(* IEC 61131-3 sources: C32_CAN/Source, 4 files *)

(* ---- ReadLocalODEntry.ST ---- *)
FUNCTION_BLOCK ReadLocalODEntry
VAR CONSTANT

    (* Definition of Data types *)
    SOO_DT_BYTE     : USINT := 1;
    SOO_DT_WORD     : USINT := 2;
    SOO_DT_DWORD    : USINT := 4;

    DEVICE          : USINT := 0;   (* Device 0: local device            *)

END_VAR

VAR_INPUT

    usiNetNumber_i  : USINT;        (* Netnumber: 0=CAN=, 1=CAN1         *)
    wIndex_i        : WORD;         (* Index to read                     *)
    bSubIndex_i     : BYTE;         (* SubIndex to read                  *)

END_VAR

VAR_OUTPUT

    dwData_o        : DWORD;        (* Data read from OD entry           *)
    usiDataType_o   : USINT;        (* DataType: 1=Byte, 2=Word, 4=Dword *)
    xSuccess_o      : BOOL;         (* TRUE if SDO was successful        *)
    wError_o        : WORD;
    dwErrorInfo_o   : DWORD;

END_VAR

VAR

    FB_CanSdoRead8  : CAN_SDO_READ8;

END_VAR

(*=========================================================================*)
(*      FUNCTIONBLOCK ReadLocalODEntry                                     *)
(*=========================================================================*)
(*                                                                         *)
(* This Function Block is used to read a numeric entry from the local      *)
(* Object Dictionary.                                                      *)
(*                                                                         *)
(* Note: This Function Block is only usable for accessing to the *LOCAL*   *)
(*       Object Dictionary. To read object entries from a remote node,     *)
(*       it is necessary to implement the complete ENABLE/CONFIRM          *)
(*       handshake procedure as described in "User Manual CANopen          *)
(*       Extension for IEC61131-3", Manual-no.: L-1008.                    *)
(*                                                                         *)
(*-------------------------------------------------------------------------*)
(*      (c) SYSTEC electronic GmbH 2009     -rs                            *)
(*=========================================================================*)

FB_CanSdoRead8 (
    NETNUMBER     := usiNetNumber_i,
    DEVICE        := DEVICE,
    INDEX         := wIndex_i,
    SUBINDEX      := bSubIndex_i,
    ENABLE        := TRUE
    |
    usiDataType_o := DATALENGTH,
    xSuccess_o    := CONFIRM,
    wError_o      := ERROR,
    dwErrorInfo_o := ERRORINFO);

FB_CanSdoRead8 (ENABLE := FALSE);

dwData_o :=             (SHL(BYTE_TO_DWORD(FB_CanSdoRead8.DATA3), 24));
dwData_o := dwData_o OR (SHL(BYTE_TO_DWORD(FB_CanSdoRead8.DATA2), 16));
dwData_o := dwData_o OR (SHL(BYTE_TO_DWORD(FB_CanSdoRead8.DATA1),  8));
dwData_o := dwData_o OR (    BYTE_TO_DWORD(FB_CanSdoRead8.DATA0)     );

RETURN;

END_FUNCTION_BLOCK

(* ---- WriteLocalODEntry.ST ---- *)
FUNCTION_BLOCK WriteLocalODEntry
VAR CONSTANT

    (* Definition of Data types *)
    SOO_DT_BYTE     : USINT := 1;
    SOO_DT_WORD     : USINT := 2;
    SOO_DT_DWORD    : USINT := 4;

    DEVICE          : USINT := 0;   (* Device 0: local device            *)

END_VAR

VAR_INPUT

    usiNetNumber_i  : USINT;        (* Netnumber: 0=CAN=, 1=CAN1         *)
    wIndex_i        : WORD;         (* Index to read                     *)
    bSubIndex_i     : BYTE;         (* SubIndex to read                  *)
    dwData_i        : DWORD;        (* Data to write into OD entry       *)
    usiDataType_i   : USINT;        (* DataType: 1=Byte, 2=Word, 4=Dword *)

END_VAR

VAR_OUTPUT

    xSuccess_o      : BOOL;         (* TRUE if SDO was successful        *)
    wError_o        : WORD;
    dwErrorInfo_o   : DWORD;

END_VAR

VAR

    FB_CanSdoWrite8 : CAN_SDO_WRITE8;

END_VAR

(*=========================================================================*)
(*      FUNCTIONBLOCK WriteLocalODEntry                                    *)
(*=========================================================================*)
(*                                                                         *)
(* This Function Block is used to write a numeric entry into the local     *)
(* Object Dictionary.                                                      *)
(*                                                                         *)
(* Note: This Function Block is only usable for accessing to the *LOCAL*   *)
(*       Object Dictionary. To write object entries into a remote node,    *)
(*       it is necessary to implement the complete ENABLE/CONFIRM          *)
(*       handshake procedure as described in "User Manual CANopen          *)
(*       Extension for IEC61131-3", Manual-no.: L-1008.                    *)
(*                                                                         *)
(*-------------------------------------------------------------------------*)
(*      (c) SYSTEC electronic GmbH 2009     -rs                            *)
(*=========================================================================*)

FB_CanSdoWrite8.DATA3 := DWORD_TO_BYTE(SHR(dwData_i, 24));
FB_CanSdoWrite8.DATA2 := DWORD_TO_BYTE(SHR(dwData_i, 16));
FB_CanSdoWrite8.DATA1 := DWORD_TO_BYTE(SHR(dwData_i,  8));
FB_CanSdoWrite8.DATA0 := DWORD_TO_BYTE(    dwData_i     );

FB_CanSdoWrite8 (
    NETNUMBER     := usiNetNumber_i,
    DEVICE        := DEVICE,
    INDEX         := wIndex_i,
    SUBINDEX      := bSubIndex_i,
    DATALENGTH    := usiDataType_i,
    ENABLE        := TRUE
    |
    xSuccess_o    := CONFIRM,
    wError_o      := ERROR,
    dwErrorInfo_o := ERRORINFO);

FB_CanSdoWrite8 (ENABLE := FALSE);

RETURN;

END_FUNCTION_BLOCK

(* ---- Main.ST ---- *)
PROGRAM Main
VAR
(***************************************************************************************************)
(************************* ShPImg variable define **************************************************)
	Functions_ShPImg 		AT %MB514.0 :BYTE;
	Modbus_connect			AT %MB515.0 :BYTE;
	ModbusAddr_ShPImg 		AT %MB516.0 :BYTE;
    Quantity_ShPImg			AT %MB517.0 :BYTE;

	TxNum					AT %MB518.0 :BYTE;

	Modbus_data0_Read		AT %MB524.0 :BYTE;
	Modbus_data1_Read		AT %MB525.0 :BYTE;
	Modbus_data2_Read		AT %MB526.0 :BYTE;
	Modbus_data3_Read		AT %MB527.0 :BYTE;
	Modbus_data4_Read		AT %MB528.0 :BYTE;
	Modbus_data5_Read		AT %MB529.0 :BYTE;
	Modbus_data6_Read		AT %MB530.0 :BYTE;
	Modbus_data7_Read		AT %MB531.0 :BYTE;
	Modbus_data8_Read		AT %MB532.0 :BYTE;
	Modbus_data9_Read		AT %MB533.0 :BYTE;

(***************************************************************************************************)
(************************* CAN variable define *****************************************************)

    bCAN1InByte0    AT %MB0.0   : BYTE;     (* mapped to Index=2000/Sub1 *)
    bCAN1InByte1    AT %MB1.0   : BYTE;     (* mapped to Index=2000/Sub2 *)
    bCAN1InByte2    AT %MB2.0   : BYTE;     (* mapped to Index=2000/Sub3 *)
    bCAN1InByte3    AT %MB3.0   : BYTE;     (* mapped to Index=2000/Sub4 *)
    bCAN1InByte4    AT %MB4.0   : BYTE;     (* mapped to Index=2000/Sub5 *)
    bCAN1InByte5    AT %MB5.0   : BYTE;     (* mapped to Index=2000/Sub6 *)
    bCAN1InByte6    AT %MB6.0   : BYTE;     (* mapped to Index=2000/Sub7 *)
    bCAN1InByte7    AT %MB7.0   : BYTE;     (* mapped to Index=2000/Sub8 *)

    bCAN1InWord0    AT %MW0.0   : WORD;     (* this overlapps 'bCAN1InByte0' and 'bCAN1InByte1' *)
    bCAN1InWord2    AT %MW2.0   : WORD;     (* this overlapps 'bCAN1InByte2' and 'bCAN1InByte3' *)
    bCAN1InWord4    AT %MW4.0   : WORD;     (* this overlapps 'bCAN1InByte4' and 'bCAN1InByte5' *)
    bCAN1InWord6    AT %MW6.0   : WORD;     (* this overlapps 'bCAN1InByte6' and 'bCAN1InByte7' *)

    bCAN1OutByte0   AT %MB256.0 : BYTE;     (* mapped to Index=2030/Sub1 *)
    bCAN1OutByte1   AT %MB257.0 : BYTE;     (* mapped to Index=2030/Sub2 *)
    bCAN1OutByte2   AT %MB258.0 : BYTE;     (* mapped to Index=2030/Sub3 *)
    bCAN1OutByte3   AT %MB259.0 : BYTE;     (* mapped to Index=2030/Sub4 *)
    bCAN1OutByte4   AT %MB260.0 : BYTE;     (* mapped to Index=2030/Sub5 *)
    bCAN1OutByte5   AT %MB261.0 : BYTE;     (* mapped to Index=2030/Sub6 *)
    bCAN1OutByte6   AT %MB262.0 : BYTE;     (* mapped to Index=2030/Sub7 *)
    bCAN1OutByte7   AT %MB263.0 : BYTE;     (* mapped to Index=2030/Sub8 *)

    wOldDataWord0                : WORD;
    wOldDataWord2                : WORD;
    wOldDataWord4                : WORD;
    wOldDataWord6                : WORD;

    udiDataCounter              : UDINT := 0;
(***************************************************************************************************)

END_VAR

(*=========================================================================*)
(*      PROGRAM Main   (used as Main Task)                                 *)
(*=========================================================================*)
(*                                                                         *)
(*-------------------------------------------------------------------------*)
(*      (c) SYSTEC electronic GmbH 2013                                    *)
(*=========================================================================*)
IF (Modbus_connect <> 1) THEN
	Functions_ShPImg := 5; (*set modbus function code*)
	ModbusAddr_ShPImg := 1; (*set modbus number of frame*)
	Modbus_connect := 1;
	Quantity_ShPImg := 8;
END_IF;

IF ((wOldDataWord0 <> bCAN1InWord0) or (wOldDataWord2 <> bCAN1InWord2)
	or (wOldDataWord4 <> bCAN1InWord4) or (wOldDataWord6 <> bCAN1InWord6)) THEN

    wOldDataWord0 := bCAN1InWord0;
    wOldDataWord2 := bCAN1InWord2;
    wOldDataWord4 := bCAN1InWord4;
    wOldDataWord6 := bCAN1InWord6;

    udiDataCounter := udiDataCounter + 1;

	Modbus_data0_Read := bCAN1InByte0;

	Modbus_data1_Read := bCAN1InByte1;

	Modbus_data2_Read := bCAN1InByte2;

	Modbus_data3_Read := bCAN1InByte3;

	Modbus_data4_Read := bCAN1InByte4;

	Modbus_data5_Read := bCAN1InByte5;

	Modbus_data6_Read := bCAN1InByte6;

	Modbus_data7_Read := bCAN1InByte7;

    TxNum := UDINT_TO_BYTE (udiDataCounter);

END_IF;

RETURN;

END_PROGRAM

(* ---- SetupCAN1.ST ---- *)
PROGRAM SetupCAN1
VAR CONSTANT

    NETNUMBER               : USINT := 1;       (* Netnumber: 0=CAN0, 1=CAN1 *)
    REMOTE_NODE_ID          : USINT := 16#40;   (* NodeID of remote node     *)

END_VAR

VAR

    FB_ReadLocalODEntry     : ReadLocalODEntry;
    FB_WriteLocalODEntry    : WriteLocalODEntry;
    udiCanID                : UDINT;
    dwCanID                 : DWORD;

END_VAR

(*=========================================================================*)
(*      PROGRAM SetupCAN1   (used as Startup Task)                         *)
(*=========================================================================*)
(*                                                                         *)
(*                                                                         *)
(*-------------------------------------------------------------------------*)
(*      (c) SYSTEC electronic GmbH 2013                                    *)
(*=========================================================================*)

(***************************************************************************)
(*                                                                         *)
(*                  Configuration of RPDO1                                 *)
(*                                                                         *)
(***************************************************************************)

(*-------------------------------------------------------------------------*)
(*  Step (1): Disable PDO by setting Bit31 in original(!) CANID            *)
(*-------------------------------------------------------------------------*)

FB_ReadLocalODEntry (
    usiNetNumber_i := NETNUMBER,
    wIndex_i       := 16#1400,      (* Index 1400:  RPDO1 communication parameter *)
    bSubIndex_i    := 1             (* SubIndex 1:  COB-ID used                   *)
    |
    dwCanID := dwData_o);

dwCanID.31 := TRUE;                 (* set Bit31 in CANID to disable the PDO      *)

FB_WriteLocalODEntry (
    usiNetNumber_i := NETNUMBER,
    wIndex_i       := 16#1400,      (* Index 1400:  RPDO1 communication parameter *)
    bSubIndex_i    := 1,            (* SubIndex 1:  COB-ID used                   *)
    dwData_i       := dwCanID,      (* CANID, marked as disabled                  *)
    usiDataType_i  := 4);           (* CANID = DWORD = 4Byte                      *)

(*-------------------------------------------------------------------------*)
(*  Step (2): Delete old mapping by setting Sub0 of PDO mapping index to 0 *)
(*-------------------------------------------------------------------------*)

FB_WriteLocalODEntry (
    usiNetNumber_i := NETNUMBER,
    wIndex_i       := 16#1600,      (* Index 1600:  RPDO1 mapping parameter       *)
    bSubIndex_i    := 0,            (* SubIndex 0:  number of mapped objects      *)
    dwData_i       := 0,            (* set number of used mapping entries to 0    *)
    usiDataType_i  := 4);           (* Sub0 = BYTE = 1Byte                        *)

(*-------------------------------------------------------------------------*)
(*  Step (3): Define new mapping of PDO                                    *)
(*-------------------------------------------------------------------------*)

FB_WriteLocalODEntry (              (* set mapping for 'CAN1InByte0'              *)
    usiNetNumber_i := NETNUMBER,
    wIndex_i       := 16#1600,      (* Index 1600:  RPDO1 mapping parameter       *)
    bSubIndex_i    := 1,            (* SubIndex 1:  1st mapped object             *)
    dwData_i       := 16#20000108,  (* Mapping:     Index=2000, Sub=01, Len=08    *)
    usiDataType_i  := 4);           (* Sub0 = DWORD = 4Byte                       *)

FB_WriteLocalODEntry (              (* set mapping for 'CAN1InByte1'              *)
    usiNetNumber_i := NETNUMBER,
    wIndex_i       := 16#1600,      (* Index 1600:  RPDO1 mapping parameter       *)
    bSubIndex_i    := 2,            (* SubIndex 2:  2st mapped object             *)
    dwData_i       := 16#20000208,  (* Mapping:     Index=2000, Sub=02, Len=08    *)
    usiDataType_i  := 4);           (* Sub0 = DWORD = 4Byte                       *)

FB_WriteLocalODEntry (              (* set mapping for 'CAN1InByte2'              *)
    usiNetNumber_i := NETNUMBER,
    wIndex_i       := 16#1600,      (* Index 1600:  RPDO1 mapping parameter       *)
    bSubIndex_i    := 3,            (* SubIndex 3:  3st mapped object             *)
    dwData_i       := 16#20000308,  (* Mapping:     Index=2000, Sub=03, Len=08    *)
    usiDataType_i  := 4);           (* Sub0 = DWORD = 4Byte                       *)

FB_WriteLocalODEntry (              (* set mapping for 'CAN1InByte3'              *)
    usiNetNumber_i := NETNUMBER,
    wIndex_i       := 16#1600,      (* Index 1600:  RPDO1 mapping parameter       *)
    bSubIndex_i    := 4,            (* SubIndex 4:  4st mapped object             *)
    dwData_i       := 16#20000408,  (* Mapping:     Index=2000, Sub=04, Len=08    *)
    usiDataType_i  := 4);           (* Sub0 = DWORD = 4Byte                       *)

FB_WriteLocalODEntry (              (* set mapping for 'CAN1InByte0'              *)
    usiNetNumber_i := NETNUMBER,
    wIndex_i       := 16#1600,      (* Index 1600:  RPDO1 mapping parameter       *)
    bSubIndex_i    := 5,            (* SubIndex 5:  5st mapped object             *)
    dwData_i       := 16#20000508,  (* Mapping:     Index=2000, Sub=05, Len=08    *)
    usiDataType_i  := 4);           (* Sub0 = DWORD = 4Byte                       *)

FB_WriteLocalODEntry (              (* set mapping for 'CAN1InByte1'              *)
    usiNetNumber_i := NETNUMBER,
    wIndex_i       := 16#1600,      (* Index 1600:  RPDO1 mapping parameter       *)
    bSubIndex_i    := 6,            (* SubIndex 6:  6st mapped object             *)
    dwData_i       := 16#20000608,  (* Mapping:     Index=2000, Sub=06, Len=08    *)
    usiDataType_i  := 4);           (* Sub0 = DWORD = 4Byte                       *)

FB_WriteLocalODEntry (              (* set mapping for 'CAN1InByte0'              *)
    usiNetNumber_i := NETNUMBER,
    wIndex_i       := 16#1600,      (* Index 1600:  RPDO1 mapping parameter       *)
    bSubIndex_i    := 7,            (* SubIndex 7:  7st mapped object             *)
    dwData_i       := 16#20000708,  (* Mapping:     Index=2000, Sub=07, Len=08    *)
    usiDataType_i  := 4);           (* Sub0 = DWORD = 4Byte                       *)

FB_WriteLocalODEntry (              (* set mapping for 'CAN1InByte1'              *)
    usiNetNumber_i := NETNUMBER,
    wIndex_i       := 16#1600,      (* Index 1600:  RPDO1 mapping parameter       *)
    bSubIndex_i    := 8,            (* SubIndex 8:  8st mapped object             *)
    dwData_i       := 16#20000808,  (* Mapping:     Index=2000, Sub=08, Len=08    *)
    usiDataType_i  := 4);           (* Sub0 = DWORD = 4Byte                       *)

(*-------------------------------------------------------------------------*)
(*  Step (4): Enable new mapping by setting number of configured objects   *)
(*-------------------------------------------------------------------------*)

FB_WriteLocalODEntry (
    usiNetNumber_i := NETNUMBER,
    wIndex_i       := 16#1600,      (* Index 1600:  RPDO1 mapping parameter       *)
    bSubIndex_i    := 0,            (* SubIndex 0:  number of mapped objects      *)
    dwData_i       := 8,            (* 1 data object (Sub1) is valid              *)
    usiDataType_i  := 1);           (* Sub0 = BYTE = 1Byte                        *)

(*-------------------------------------------------------------------------*)
(*  Step (5): Enable PDO by setting valid (new) CANID                      *)
(*-------------------------------------------------------------------------*)

dwCanID := USINT_TO_DWORD(REMOTE_NODE_ID) OR 16#00000180;

FB_WriteLocalODEntry (
    usiNetNumber_i := NETNUMBER,
    wIndex_i       := 16#1400,      (* Index 1400:  RPDO1 communication parameter *)
    bSubIndex_i    := 1,            (* SubIndex 1:  COB-ID used                   *)
    dwData_i       := dwCanID,      (* CANID, marked as enabled                   *)
    usiDataType_i  := 4);           (* CANID = DWORD = 4Byte                      *)

(***************************************************************************)
(*                                                                         *)
(*                  Configuration of TPDO1                                 *)
(*                                                                         *)
(***************************************************************************)

(*-------------------------------------------------------------------------*)
(*  Step (1): Disable PDO by setting Bit31 in original(!) CANID            *)
(*-------------------------------------------------------------------------*)

FB_ReadLocalODEntry (
    usiNetNumber_i := NETNUMBER,
    wIndex_i       := 16#1800,      (* Index 1800:  TPDO1 communication parameter *)
    bSubIndex_i    := 1             (* SubIndex 1:  COB-ID used                   *)
    |
    dwCanID := dwData_o);

dwCanID.31 := TRUE;                 (* set Bit31 in CANID to disable the PDO      *)

FB_WriteLocalODEntry (
    usiNetNumber_i := NETNUMBER,
    wIndex_i       := 16#1800,      (* Index 1800:  TPDO1 communication parameter *)
    bSubIndex_i    := 1,            (* SubIndex 1:  COB-ID used                   *)
    dwData_i       := dwCanID,      (* CANID, marked as disabled                  *)
    usiDataType_i  := 4);           (* CANID = DWORD = 4Byte                      *)

(*-------------------------------------------------------------------------*)
(*  Step (2): Delete old mapping by setting Sub0 of PDO mapping index to 0 *)
(*-------------------------------------------------------------------------*)

FB_WriteLocalODEntry (
    usiNetNumber_i := NETNUMBER,
    wIndex_i       := 16#1A00,      (* Index 1A00:  TPDO1 mapping parameter       *)
    bSubIndex_i    := 0,            (* SubIndex 0:  number of mapped objects      *)
    dwData_i       := 0,            (* set number of used mapping entries to 0    *)
    usiDataType_i  := 1);           (* Sub0 = BYTE = 1Byte                        *)

(*-------------------------------------------------------------------------*)
(*  Step (3): Define new mapping of PDO                                    *)
(*-------------------------------------------------------------------------*)

FB_WriteLocalODEntry (              (* set mapping for 'CAN1OutByte0'             *)
    usiNetNumber_i := NETNUMBER,
    wIndex_i       := 16#1A00,      (* Index 1A00:  TPDO1 mapping parameter       *)
    bSubIndex_i    := 1,            (* SubIndex 1:  1st mapped object             *)
    dwData_i       := 16#20300108,  (* Mapping:     Index=2030, Sub=01, Len=08    *)
    usiDataType_i  := 4);           (* Sub0 = DWORD = 4Byte                       *)

FB_WriteLocalODEntry (              (* set mapping for 'CAN1InByte1'              *)
    usiNetNumber_i := NETNUMBER,
    wIndex_i       := 16#1A00,      (* Index 1600:  RPDO1 mapping parameter       *)
    bSubIndex_i    := 2,            (* SubIndex 2:  2nd mapped object             *)
    dwData_i       := 16#20300208,  (* Mapping:     Index=2030, Sub=02, Len=08    *)
    usiDataType_i  := 4);           (* Sub0 = DWORD = 4Byte                       *)

FB_WriteLocalODEntry (              (* set mapping for 'CAN1OutByte2'             *)
    usiNetNumber_i := NETNUMBER,
    wIndex_i       := 16#1A00,      (* Index 1A00:  TPDO1 mapping parameter       *)
    bSubIndex_i    := 3,            (* SubIndex 3:  1st mapped object             *)
    dwData_i       := 16#20300308,  (* Mapping:     Index=2030, Sub=03, Len=08    *)
    usiDataType_i  := 4);           (* Sub0 = DWORD = 4Byte                       *)

FB_WriteLocalODEntry (              (* set mapping for 'CAN1OutByte0'             *)
    usiNetNumber_i := NETNUMBER,
    wIndex_i       := 16#1A00,      (* Index 1A00:  TPDO1 mapping parameter       *)
    bSubIndex_i    := 4,            (* SubIndex 4:  1st mapped object             *)
    dwData_i       := 16#20300408,  (* Mapping:     Index=2030, Sub=04, Len=08    *)
    usiDataType_i  := 4);           (* Sub0 = DWORD = 4Byte                       *)

FB_WriteLocalODEntry (              (* set mapping for 'CAN1InByte1'              *)
    usiNetNumber_i := NETNUMBER,
    wIndex_i       := 16#1A00,      (* Index 1600:  RPDO1 mapping parameter       *)
    bSubIndex_i    := 5,            (* SubIndex 5:  2nd mapped object             *)
    dwData_i       := 16#20300508,  (* Mapping:     Index=2030, Sub=05, Len=08    *)
    usiDataType_i  := 4);           (* Sub0 = DWORD = 4Byte                       *)

FB_WriteLocalODEntry (              (* set mapping for 'CAN1OutByte2'             *)
    usiNetNumber_i := NETNUMBER,
    wIndex_i       := 16#1A00,      (* Index 1A00:  TPDO1 mapping parameter       *)
    bSubIndex_i    := 6,            (* SubIndex 6:  1st mapped object             *)
    dwData_i       := 16#20300608,  (* Mapping:     Index=2030, Sub=06, Len=08    *)
    usiDataType_i  := 4);           (* Sub0 = DWORD = 4Byte                       *)

FB_WriteLocalODEntry (              (* set mapping for 'CAN1OutByte0'             *)
    usiNetNumber_i := NETNUMBER,
    wIndex_i       := 16#1A00,      (* Index 1A00:  TPDO1 mapping parameter       *)
    bSubIndex_i    := 7,            (* SubIndex 7:  1st mapped object             *)
    dwData_i       := 16#20300708,  (* Mapping:     Index=2030, Sub=07, Len=08    *)
    usiDataType_i  := 4);           (* Sub0 = DWORD = 4Byte                       *)

FB_WriteLocalODEntry (              (* set mapping for 'CAN1InByte1'              *)
    usiNetNumber_i := NETNUMBER,
    wIndex_i       := 16#1A00,      (* Index 1600:  RPDO1 mapping parameter       *)
    bSubIndex_i    := 8,            (* SubIndex 8:  2nd mapped object             *)
    dwData_i       := 16#20300808,  (* Mapping:     Index=2030, Sub=08, Len=08    *)
    usiDataType_i  := 4);           (* Sub0 = DWORD = 4Byte                       *)

(*-------------------------------------------------------------------------*)
(*  Step (4): Enable new mapping by setting number of configured objects   *)
(*-------------------------------------------------------------------------*)

FB_WriteLocalODEntry (
    usiNetNumber_i := NETNUMBER,
    wIndex_i       := 16#1A00,      (* Index 1A00:  TPDO1 mapping parameter       *)
    bSubIndex_i    := 0,            (* SubIndex 0:  number of mapped objects      *)
    dwData_i       := 8,            (* 2 data objects (Sub1+Sub2) are valid       *)
    usiDataType_i  := 1);           (* Sub0 = BYTE = 1Byte                        *)

(*-------------------------------------------------------------------------*)
(*  Step (5): Enable PDO by setting valid CANID                            *)
(*-------------------------------------------------------------------------*)

udiCanID := 16#00000200 + USINT_TO_UDINT(REMOTE_NODE_ID);
dwCanID := UDINT_TO_DWORD(udiCanID);

FB_WriteLocalODEntry (
    usiNetNumber_i := NETNUMBER,
    wIndex_i       := 16#1800,      (* Index 1800:  TPDO1 communication parameter *)
    bSubIndex_i    := 1,            (* SubIndex 1:  COB-ID used                   *)
    dwData_i       := dwCanID,      (* CANID, marked as enabled                   *)
    usiDataType_i  := 4);           (* CANID = DWORD = 4Byte                      *)

RETURN;

END_PROGRAM
